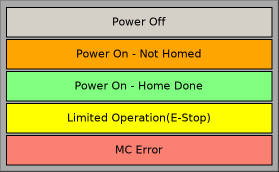
VISUALIZATION vis_Axis_Control_Backgroud_Descripton  // 279x172
    Rectangle (0,0 279x172)
    Rectangle (6,7 266x30), "Power Off"
    Rectangle (6,71 266x30), "Power On - Home Done"
    Rectangle (6,103 266x30), "Limited Operation(E-Stop)"
    Rectangle (6,135 266x30), "MC Error"
    Rectangle (6,39 266x30), "Power On - Not Homed"
END_VISUALIZATION

(* stored: Version 1.1.0.1, ProductVersion 3.1.4024.12
   Visu vis_Axis_Control_Backgroud_Descripton: Id {bc6fcdcc-374b-4708-9801-be98ddffa527} *)
